// TIA Portal V16 export
// export: Created 2022-07-21T09:35:35.1718284Z, ExportSetting WithDefaults, DisplayName Totally Integrated Automation Portal, DisplayVersion V16 Update 4, DisplayName TIA Portal Version Control Interface, DisplayVersion V16 Update 2, DisplayName TIA Portal Openness, DisplayVersion V16 Update 4, DisplayName SINAMICS Startdrive Advanced, DisplayVersion V16 Update 5, DisplayName SINAMICS Startdrive G130, G150, S120, S150, SINAMICS MV, S210, DisplayVersion V16 Update 5, DisplayName SINAMICS Startdrive G110M, G120, G120C, G120D, G120P, G115D, DisplayVersion V16 Update 5, DisplayName STEP 7 Professional, DisplayVersion V16 Update 4, DisplayName STEP 7 Safety, DisplayVersion V16, DisplayName WinCC Advanced, DisplayVersion V16 Update 4
FUNCTION_BLOCK "fbKRC4ExtAut"   // FB30, LAD
TITLE = External automation handling for KUKA KRC4 / Blok obsługi trybu automatyki zewnętrznej KUKA KRC4
{ S7_Optimized_Access := 'TRUE' }
VERSION : 0.1
// stored: AutoNumber false, IsIECCheckEnabled false, IsRetainMemResEnabled false, MemoryReserve 100, SetENOAutomatically false, UDAEnableTagReadback false
   VAR_INPUT
      inRobotOutputs : "typeKRC4Outputs";   // Wejścia standardowe robota / Robot standard inputs
      inAuto : Bool;   // Zezwolenie ogólne dla robota na ruch w trybie automatycznym / Enable movement in automatic mode
      inExtReset : Bool;   // Żądanie kasowania błędów / Alarm reset requested
      inStart : Bool;   // Start programu zadanego przez PgNo / Start program selected by PgNo
      inPgNo : USInt;   // Numer programu do startu w trybie automatycznym / Program number to start in automatic mode
      inServicePos : Bool;   // Robot w poyzcji serwisowej / Robot in service position
      inClock : Bool;   // Bit zegara systemowego dla generowania zbocza sygnału / Memory clock bit for signal edge generation
   END_VAR
   VAR_OUTPUT
      ouRobotInputs : "typeKRC4Inputs";   // Wyjścia standardowe robota / Robot standard outputs
      ouStdProgSelected : Bool;   // Wybrano program standardowy / Standard program selected
      ouHomePosSelected { ExternalAccessible := 'False'; ExternalVisible := 'False'; ExternalWritable := 'False'} : Bool;   // Wybrano program "pozycja bazowa" / Home position program selected
      ouServicePosSelected { ExternalAccessible := 'False'; ExternalVisible := 'False'; ExternalWritable := 'False'} : Bool;   // Wybrano program "pozycja serwisowa" / Service position program selected
      ouBrakeTestSelected { ExternalAccessible := 'False'; ExternalVisible := 'False'; ExternalWritable := 'False'} : Bool;   // Wybrano program "test hamulców" / Brake test program selected
      ouMasterTestSelected { ExternalAccessible := 'False'; ExternalVisible := 'False'; ExternalWritable := 'False'} : Bool;   // Wybrano program "test referencji" / Reference test program selected
   END_VAR
   VAR_IN_OUT
      ioRobot : "typeRobot";
   END_VAR
   VAR
      sTONIntReset { ExternalAccessible := 'False'; ExternalVisible := 'False'; ExternalWritable := 'False'} : IEC_TIMER;   // Wewnętrzny reset (timer) / Internal reset (timer)
      sTOFHoldReset { ExternalAccessible := 'False'; ExternalVisible := 'False'; ExternalWritable := 'False'} : IEC_TIMER;   // Podtrzymanie wewnętrznego resetu (timer) / Hold internal reset (timer)
      sTONPgNoValDly { ExternalAccessible := 'False'; ExternalVisible := 'False'; ExternalWritable := 'False'} : IEC_TIMER;   // Numer programu prawidłowy (timer) / Correct program number (timer)
      sSIntPgNoPrevCycle { ExternalAccessible := 'False'; ExternalVisible := 'False'; ExternalWritable := 'False'} : USInt;   // Numer programu z poprzedniego cyklu / Previous cycle program number
      sBoPFlk { ExternalAccessible := 'False'; ExternalVisible := 'False'; ExternalWritable := 'False'} : Array[1..15] of Bool;   // Bity dla wykrywania zbocza / Edge detection bits
      sBoAutoRdy { ExternalWritable := 'False'} : Bool;   // Robot gotowy do pracy w trybie automatyki zewnętrznej / Robot ready to work in external automation mode
      sBoPgNoValid { ExternalWritable := 'False'} : Bool;   // Numer programu prawidłowy / Correct program number
      sBoExtStart { ExternalWritable := 'False'} : Bool;   // Zewnętrzny start lub kontynuacja programu / External start/continue program
      sBoMoveEnable { ExternalWritable := 'False'} : Bool;   // Ogólne zezwolenie na ruch / Movement enable
      sBoPgReset { ExternalWritable := 'False'} : Bool;   // Automatyczny reset programu / Automatic program reset
      sBoReadyForProgram { ExternalWritable := 'False'} : Bool;   // Robot gotowy do przyjęcia programu / Robot ready to receive new program
      instReset { S7_SetPoint := 'True'} : "fbReset";
   END_VAR
   VAR_TEMP
      tTrue : Bool;   // Zawsze "prawda" / Always true
      tFalse : Bool;   // Zawsze "fałsz" / Always false
      tIntResetTrigger : Bool;   // Wyzwolenie wewnętrznego resetu / Trigger internal reset
      tIntReset : Bool;   // Żądanie wewnętrznego resetu / External reset requested
      tPgNoValidDly : Bool;   // Numer programu prawidłowy (opóźniony) / Correct program number (delayed)
      tRobotInServicePosition : Bool;
   END_VAR
   VAR_TEMP   // added for the SCL form of the ladder/FBD networks
      _w1 : Bool;
      _w2 : Bool;
      _w3 : Bool;
      _w4 : Bool;
   END_VAR
BEGIN

REGION Network 1: Information / Informacja
   // EXT mode handling for KUKA KRC4 robots with brake test and reference test.
   // * Used inputs: 22
   // * Used outputs: 32
   // * Variables configuration for external automation:
   // -PGNO_TYPE = 1
   // -REFLECT_PROG_NR = 1
   // -PGNO_LENGTH = 8 (bits)
   // * Input adresses configuration in robot: as in "typeKRCInputs"
   // * Output adresses configuration in robot: as in "typeKRCOutputs"
   // 
   // !!! WARNING !!! Specify program numbers in controller constants: 
   // Robot.PgNoBrakeTest 
   // Robot.PgNoMasterTest
   // Robot.PgNoServicePos
   // Obsługa trybu EXT robotów KUKA KRC4 z obsługą testu hamulców i referencji.
   // * Liczba użwanych wejść: 22
   // * Liczba używanych wyjść: 32
   // * Konfiguracja zmiennych dla automatyki zewnętrznej:
   // - PGNO_TYPE = 1
   // - REFLECT_PROG_NR = 1
   // - PGNO_LENGTH = 8 (bitow)
   // * Konfiguracja adresów wejść w robocie: tak jak "typeKRCInputs"
   // * Konfiguracja adresów wyjść w robocie: tak jak "typeKRCOutputs"
   // 
   // !!! UWAGA !!!Należy podać numery programów w w stałych sterownika:
   // Robot.PgNoBrakeTest - test hamulców
   // Robot.PgNoMasterTest - test masteringu
   // Robot.PgNoServicePos - dojazd do pozycji serwisowej
END_REGION

REGION Network 2: Always true / Zawsze "prawda"
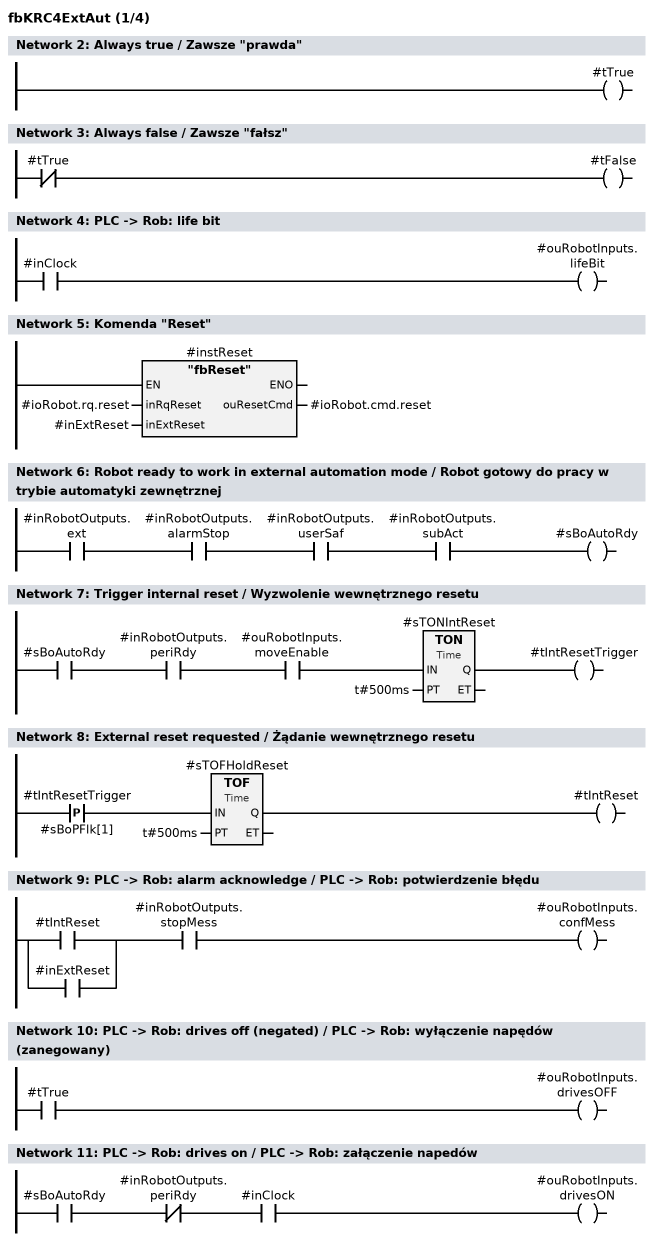
   RUNG wire#powerrail
      Coil( #tTrue )
   END_RUNG
   // the same network as SCL:
   #tTrue := TRUE;
END_REGION

REGION Network 3: Always false / Zawsze "fałsz"
   RUNG wire#powerrail
      I_Contact( #tTrue )
      Coil( #tFalse )
   END_RUNG
   // the same network as SCL:
   #tFalse := NOT #tTrue;
END_REGION

REGION Network 4: PLC -> Rob: life bit
   RUNG wire#powerrail
      Contact( #inClock )
      Coil( #ouRobotInputs.lifeBit )
   END_RUNG
   // the same network as SCL:
   #ouRobotInputs.lifeBit := #inClock;
END_REGION

REGION Network 5: Komenda "Reset"
   RUNG wire#powerrail
      #instReset(inRqReset := #ioRobot.rq.reset, inExtReset := #inExtReset, ouResetCmd => #ioRobot.cmd.reset)
   END_RUNG
   // the same network as SCL:
   #instReset(inRqReset := #ioRobot.rq.reset, inExtReset := #inExtReset, ouResetCmd => #ioRobot.cmd.reset);   // "fbReset"
END_REGION

REGION Network 6: Robot ready to work in external automation mode / Robot gotowy do pracy w trybie automatyki zewnętrznej
   RUNG wire#powerrail
      Contact( #inRobotOutputs.ext )
      Contact( #inRobotOutputs.alarmStop )
      Contact( #inRobotOutputs.userSaf )
      Contact( #inRobotOutputs.subAct )
      Coil( #sBoAutoRdy )
   END_RUNG
   // the same network as SCL:
   #sBoAutoRdy := #inRobotOutputs.ext AND #inRobotOutputs.alarmStop AND #inRobotOutputs.userSaf AND #inRobotOutputs.subAct;
END_REGION

REGION Network 7: Trigger internal reset / Wyzwolenie wewnętrznego resetu
   RUNG wire#powerrail
      Contact( #sBoAutoRdy )
      Contact( #inRobotOutputs.periRdy )
      Contact( #ouRobotInputs.moveEnable )
      { S7_Templates := "time_type := Time" } #sTONIntReset.TON(pt := t#500ms, et =>)
      Coil( #tIntResetTrigger )
   END_RUNG
   // the same network as SCL:
   #sTONIntReset.TON(IN := #sBoAutoRdy AND #inRobotOutputs.periRdy AND #ouRobotInputs.moveEnable, PT := t#500ms);
   #tIntResetTrigger := #sTONIntReset.Q;
END_REGION

REGION Network 8: External reset requested / Żądanie wewnętrznego resetu
   RUNG wire#powerrail
      P_Contact(operand := #tIntResetTrigger, bit := #sBoPFlk[1])
      { S7_Templates := "time_type := Time" } #sTOFHoldReset.TOF(pt := t#500ms, et =>)
      Coil( #tIntReset )
   END_RUNG
   // the same network as SCL:
   #_w1 := #tIntResetTrigger AND NOT #sBoPFlk[1];   // rising edge of #tIntResetTrigger
   #sBoPFlk[1] := #tIntResetTrigger;
   #sTOFHoldReset.TOF(IN := #_w1, PT := t#500ms);
   #tIntReset := #sTOFHoldReset.Q;
END_REGION

REGION Network 9: PLC -> Rob: alarm acknowledge / PLC -> Rob: potwierdzenie błędu
   RUNG wire#powerrail
      Contact( #tIntReset )
      wire#w1
      Contact( #inRobotOutputs.stopMess )
      Coil( #ouRobotInputs.confMess )
   END_RUNG
   RUNG wire#powerrail
      Contact( #inExtReset )
   END_RUNG wire#w1
   // the same network as SCL:
   #ouRobotInputs.confMess := (#tIntReset OR #inExtReset) AND #inRobotOutputs.stopMess;
END_REGION

REGION Network 10: PLC -> Rob: drives off (negated) / PLC -> Rob: wyłączenie napędów (zanegowany)
   RUNG wire#powerrail
      Contact( #tTrue )
      Coil( #ouRobotInputs.drivesOFF )
   END_RUNG
   // the same network as SCL:
   #ouRobotInputs.drivesOFF := #tTrue;
END_REGION

REGION Network 11: PLC -> Rob: drives on / PLC -> Rob: załączenie napedów
   RUNG wire#powerrail
      Contact( #sBoAutoRdy )
      I_Contact( #inRobotOutputs.periRdy )
      Contact( #inClock )
      Coil( #ouRobotInputs.drivesON )
   END_RUNG
   // the same network as SCL:
   #ouRobotInputs.drivesON := #sBoAutoRdy AND NOT #inRobotOutputs.periRdy AND #inClock;
END_REGION

REGION Network 12: PLC -> Rob: external start program / PLC -> Rob: zewnętrzny start programu
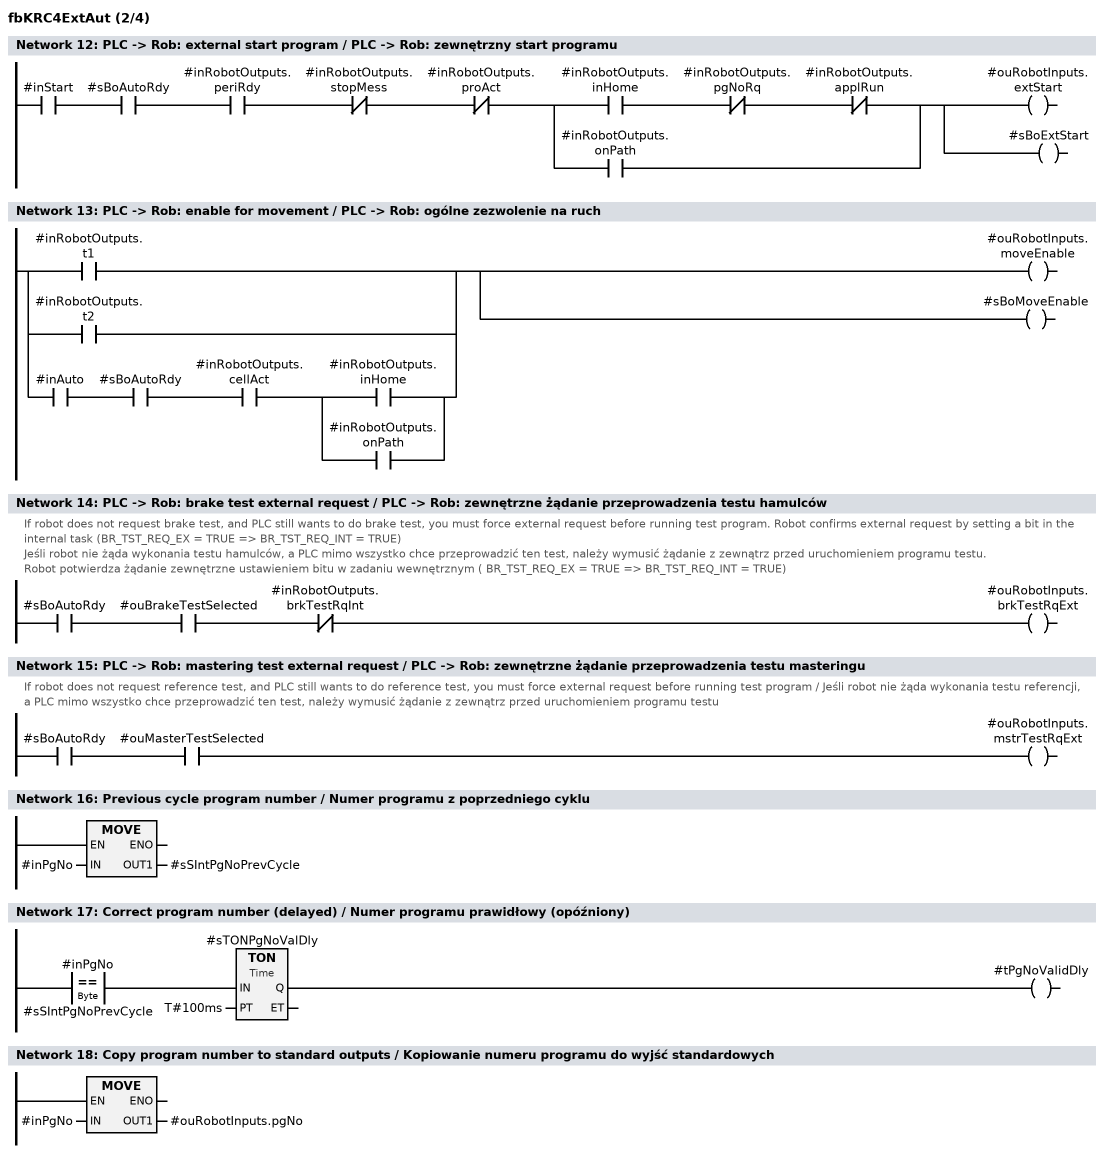
   RUNG wire#powerrail
      Contact( #inStart )
      Contact( #sBoAutoRdy )
      Contact( #inRobotOutputs.periRdy )
      I_Contact( #inRobotOutputs.stopMess )
      I_Contact( #inRobotOutputs.proAct )
      wire#w1
      Contact( #inRobotOutputs.inHome )
      I_Contact( #inRobotOutputs.pgNoRq )
      I_Contact( #inRobotOutputs.applRun )
      wire#w2
      Coil( #ouRobotInputs.extStart )
   END_RUNG
   RUNG wire#w1
      Contact( #inRobotOutputs.onPath )
   END_RUNG wire#w2
   RUNG wire#w2
      Coil( #sBoExtStart )
   END_RUNG
   // the same network as SCL:
   #ouRobotInputs.extStart := #inStart AND #sBoAutoRdy AND #inRobotOutputs.periRdy AND NOT #inRobotOutputs.stopMess AND NOT #inRobotOutputs.proAct AND ((#inRobotOutputs.inHome AND NOT #inRobotOutputs.pgNoRq AND NOT #inRobotOutputs.applRun) OR #inRobotOutputs.onPath);
   #sBoExtStart := #ouRobotInputs.extStart;
END_REGION

REGION Network 13: PLC -> Rob: enable for movement / PLC -> Rob: ogólne zezwolenie na ruch
   RUNG wire#powerrail
      Contact( #inRobotOutputs.t1 )
      wire#w1
      Coil( #ouRobotInputs.moveEnable )
   END_RUNG
   RUNG wire#powerrail
      Contact( #inRobotOutputs.t2 )
   END_RUNG wire#w1
   RUNG wire#powerrail
      Contact( #inAuto )
      Contact( #sBoAutoRdy )
      Contact( #inRobotOutputs.cellAct )
      wire#w2
      Contact( #inRobotOutputs.inHome )
   END_RUNG wire#w1
   RUNG wire#w2
      Contact( #inRobotOutputs.onPath )
   END_RUNG wire#w1
   RUNG wire#w1
      Coil( #sBoMoveEnable )
   END_RUNG
   // the same network as SCL:
   #ouRobotInputs.moveEnable := #inRobotOutputs.t1 OR #inRobotOutputs.t2 OR (#inAuto AND #sBoAutoRdy AND #inRobotOutputs.cellAct AND (#inRobotOutputs.inHome OR #inRobotOutputs.onPath));
   #sBoMoveEnable := #ouRobotInputs.moveEnable;
END_REGION

REGION Network 14: PLC -> Rob: brake test external request / PLC -> Rob: zewnętrzne żądanie przeprowadzenia testu hamulców
   // If robot does not request brake test, and PLC still wants to do brake test, you must force external request before running test program. Robot confirms external request by setting a bit in the internal task (BR_TST_REQ_EX = TRUE => BR_TST_REQ_INT = TRUE)
   // Jeśli robot nie żąda wykonania testu hamulców, a PLC mimo wszystko chce przeprowadzić ten test, należy wymusić żądanie z zewnątrz przed uruchomieniem programu testu.
   // Robot potwierdza żądanie zewnętrzne ustawieniem bitu w zadaniu wewnętrznym ( BR_TST_REQ_EX = TRUE => BR_TST_REQ_INT = TRUE)
   RUNG wire#powerrail
      Contact( #sBoAutoRdy )
      Contact( #ouBrakeTestSelected )
      I_Contact( #inRobotOutputs.brkTestRqInt )
      Coil( #ouRobotInputs.brkTestRqExt )
   END_RUNG
   // the same network as SCL:
   #ouRobotInputs.brkTestRqExt := #sBoAutoRdy AND #ouBrakeTestSelected AND NOT #inRobotOutputs.brkTestRqInt;
END_REGION

REGION Network 15: PLC -> Rob: mastering test external request / PLC -> Rob: zewnętrzne żądanie przeprowadzenia testu masteringu
   // If robot does not request reference test, and PLC still wants to do reference test, you must force external request before running test program / Jeśli robot nie żąda wykonania testu referencji, a PLC mimo wszystko chce przeprowadzić ten test, należy wymusić żądanie z zewnątrz przed uruchomieniem programu testu
   RUNG wire#powerrail
      Contact( #sBoAutoRdy )
      Contact( #ouMasterTestSelected )
      Coil( #ouRobotInputs.mstrTestRqExt )
   END_RUNG
   // the same network as SCL:
   #ouRobotInputs.mstrTestRqExt := #sBoAutoRdy AND #ouMasterTestSelected;
END_REGION

REGION Network 16: Previous cycle program number / Numer programu z poprzedniego cyklu
   RUNG wire#powerrail
      Move(in := #inPgNo, out1 => #sSIntPgNoPrevCycle)
   END_RUNG
   // the same network as SCL:
   #sSIntPgNoPrevCycle := #inPgNo;
END_REGION

REGION Network 17: Correct program number (delayed) / Numer programu prawidłowy (opóźniony)
   RUNG wire#powerrail
      { S7_Templates := "SrcType := Byte" } EQ_Contact(in1 := #inPgNo, in2 := #sSIntPgNoPrevCycle)
      { S7_Templates := "time_type := Time" } #sTONPgNoValDly.TON(pt := T#100ms, et =>)
      Coil( #tPgNoValidDly )
   END_RUNG
   // the same network as SCL:
   #sTONPgNoValDly.TON(IN := #inPgNo = #sSIntPgNoPrevCycle, PT := T#100ms);
   #tPgNoValidDly := #sTONPgNoValDly.Q;
END_REGION

REGION Network 18: Copy program number to standard outputs / Kopiowanie numeru programu do wyjść standardowych
   RUNG wire#powerrail
      Move(in := #inPgNo, out1 => #ouRobotInputs.pgNo)
   END_RUNG
   // the same network as SCL:
   #ouRobotInputs.pgNo := #inPgNo;
END_REGION

REGION Network 19: PLC -> Rob: program number - correct / PLC -> Rob: nr programu - poprawny
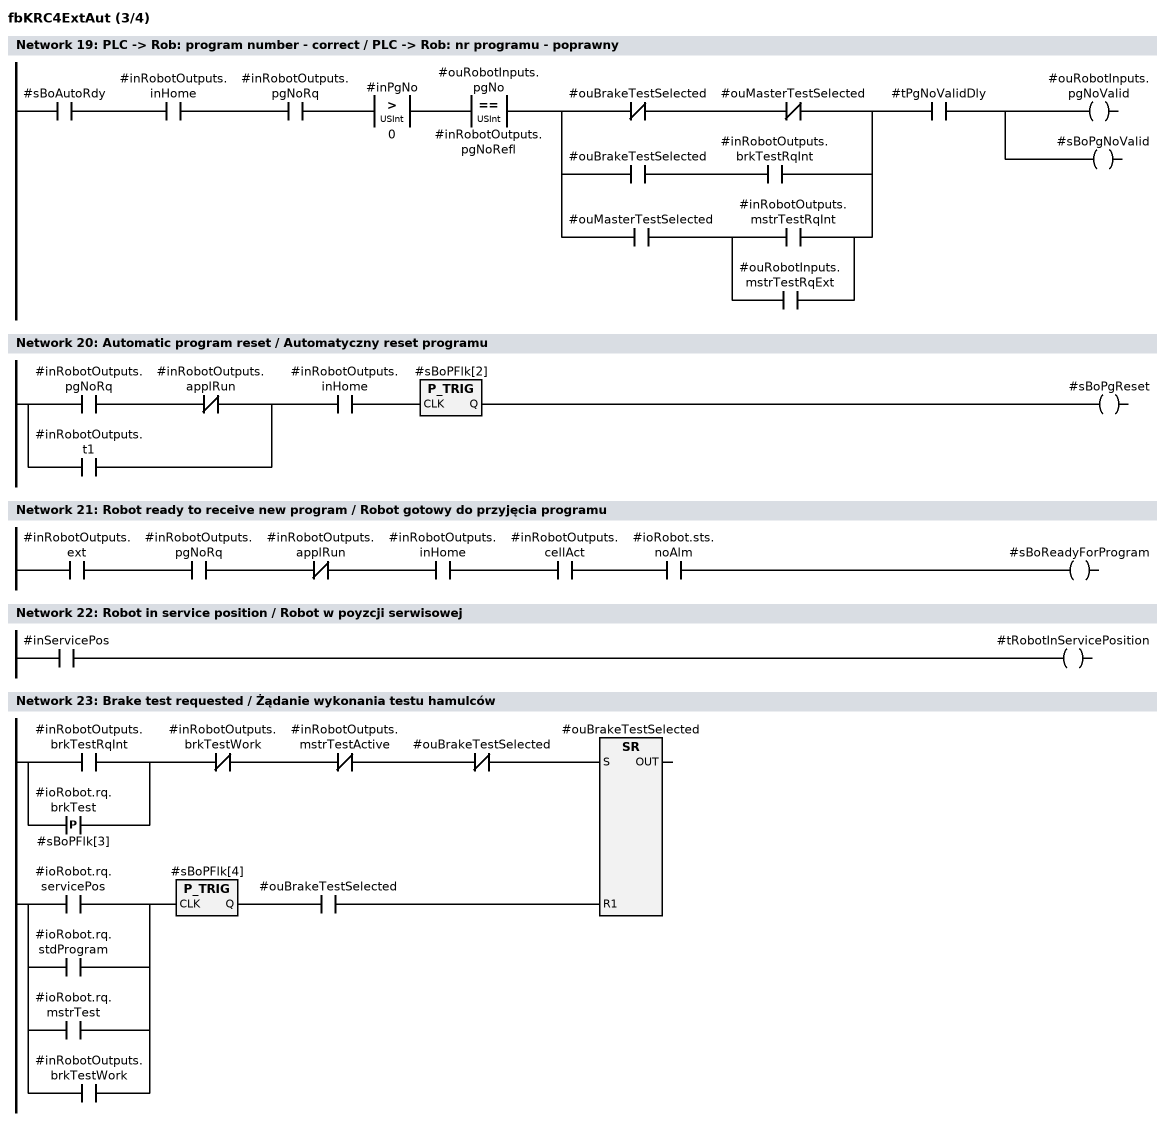
   RUNG wire#powerrail
      Contact( #sBoAutoRdy )
      Contact( #inRobotOutputs.inHome )
      Contact( #inRobotOutputs.pgNoRq )
      { S7_Templates := "SrcType := USInt" } GT_Contact(in1 := #inPgNo, in2 := 0)
      { S7_Templates := "SrcType := USInt" } EQ_Contact(in1 := #ouRobotInputs.pgNo, in2 := #inRobotOutputs.pgNoRefl)
      wire#w1
      I_Contact( #ouBrakeTestSelected )
      I_Contact( #ouMasterTestSelected )
      wire#w2
      Contact( #tPgNoValidDly )
      wire#w4
      Coil( #ouRobotInputs.pgNoValid )
   END_RUNG
   RUNG wire#w1
      Contact( #ouBrakeTestSelected )
      Contact( #inRobotOutputs.brkTestRqInt )
   END_RUNG wire#w2
   RUNG wire#w1
      Contact( #ouMasterTestSelected )
      wire#w3
      Contact( #inRobotOutputs.mstrTestRqInt )
   END_RUNG wire#w2
   RUNG wire#w3
      Contact( #ouRobotInputs.mstrTestRqExt )
   END_RUNG wire#w2
   RUNG wire#w4
      Coil( #sBoPgNoValid )
   END_RUNG
   // the same network as SCL:
   #ouRobotInputs.pgNoValid := #sBoAutoRdy AND #inRobotOutputs.inHome AND #inRobotOutputs.pgNoRq AND (#inPgNo > 0) AND (#ouRobotInputs.pgNo = #inRobotOutputs.pgNoRefl) AND ((NOT #ouBrakeTestSelected AND NOT #ouMasterTestSelected) OR (#ouBrakeTestSelected AND #inRobotOutputs.brkTestRqInt) OR (#ouMasterTestSelected AND (#inRobotOutputs.mstrTestRqInt OR #ouRobotInputs.mstrTestRqExt))) AND #tPgNoValidDly;
   #sBoPgNoValid := #ouRobotInputs.pgNoValid;
END_REGION

REGION Network 20: Automatic program reset / Automatyczny reset programu
   RUNG wire#powerrail
      Contact( #inRobotOutputs.pgNoRq )
      I_Contact( #inRobotOutputs.applRun )
      wire#w1
      Contact( #inRobotOutputs.inHome )
      P_Trig( #sBoPFlk[2] )
      Coil( #sBoPgReset )
   END_RUNG
   RUNG wire#powerrail
      Contact( #inRobotOutputs.t1 )
   END_RUNG wire#w1
   // the same network as SCL:
   #_w1 := ((#inRobotOutputs.pgNoRq AND NOT #inRobotOutputs.applRun) OR #inRobotOutputs.t1) AND #inRobotOutputs.inHome;
   #_w2 := #_w1 AND NOT #sBoPFlk[2];   // rising edge
   #sBoPFlk[2] := #_w1;
   #sBoPgReset := #_w2;
END_REGION

REGION Network 21: Robot ready to receive new program / Robot gotowy do przyjęcia programu
   RUNG wire#powerrail
      Contact( #inRobotOutputs.ext )
      Contact( #inRobotOutputs.pgNoRq )
      I_Contact( #inRobotOutputs.applRun )
      Contact( #inRobotOutputs.inHome )
      Contact( #inRobotOutputs.cellAct )
      Contact( #ioRobot.sts.noAlm )
      Coil( #sBoReadyForProgram )
   END_RUNG
   // the same network as SCL:
   #sBoReadyForProgram := #inRobotOutputs.ext AND #inRobotOutputs.pgNoRq AND NOT #inRobotOutputs.applRun AND #inRobotOutputs.inHome AND #inRobotOutputs.cellAct AND #ioRobot.sts.noAlm;
END_REGION

REGION Network 22: Robot in service position / Robot w poyzcji serwisowej
   RUNG wire#powerrail
      Contact( #inServicePos )
      Coil( #tRobotInServicePosition )
   END_RUNG
   // the same network as SCL:
   #tRobotInServicePosition := #inServicePos;
END_REGION

REGION Network 23: Brake test requested / Żądanie wykonania testu hamulców
   RUNG wire#powerrail
      Contact( #inRobotOutputs.brkTestRqInt )
      wire#w1
      I_Contact( #inRobotOutputs.brkTestWork )
      I_Contact( #inRobotOutputs.mstrTestActive )
      I_Contact( #ouBrakeTestSelected )
      S_SR(operand := #ouBrakeTestSelected, r1 := wire#w3)
   END_RUNG
   RUNG wire#powerrail
      P_Contact(operand := #ioRobot.rq.brkTest, bit := #sBoPFlk[3])
   END_RUNG wire#w1
   RUNG wire#powerrail
      Contact( #ioRobot.rq.servicePos )
      wire#w2
      P_Trig( #sBoPFlk[4] )
      Contact( #ouBrakeTestSelected )
   END_RUNG wire#w3
   RUNG wire#powerrail
      Contact( #ioRobot.rq.stdProgram )
   END_RUNG wire#w2
   RUNG wire#powerrail
      Contact( #ioRobot.rq.mstrTest )
   END_RUNG wire#w2
   RUNG wire#powerrail
      Contact( #inRobotOutputs.brkTestWork )
   END_RUNG wire#w2
   // the same network as SCL:
   #_w1 := #ioRobot.rq.brkTest AND NOT #sBoPFlk[3];   // rising edge of #ioRobot.rq.brkTest
   #sBoPFlk[3] := #ioRobot.rq.brkTest;
   #_w2 := #ioRobot.rq.servicePos OR #ioRobot.rq.stdProgram OR #ioRobot.rq.mstrTest OR #inRobotOutputs.brkTestWork;
   #_w3 := #_w2 AND NOT #sBoPFlk[4];   // rising edge
   #sBoPFlk[4] := #_w2;
   #_w4 := #_w3 AND #ouBrakeTestSelected;
   IF (#inRobotOutputs.brkTestRqInt OR #_w1) AND NOT #inRobotOutputs.brkTestWork AND NOT #inRobotOutputs.mstrTestActive AND NOT #ouBrakeTestSelected THEN
       #ouBrakeTestSelected := TRUE;   // SR flip-flop
   END_IF;
   IF #_w4 THEN #ouBrakeTestSelected := FALSE; END_IF;
END_REGION

REGION Network 24: Robot 1 request mastering test / Robot 1 żądanie wykonania testu masteringu
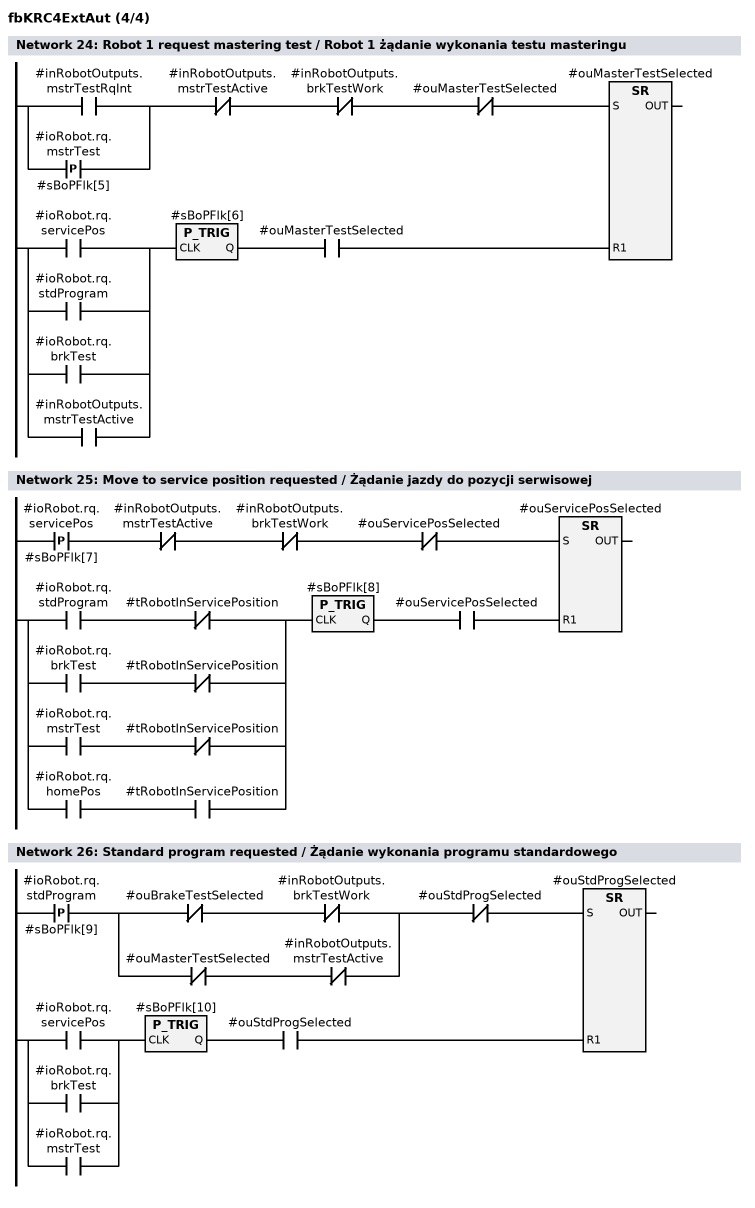
   RUNG wire#powerrail
      Contact( #inRobotOutputs.mstrTestRqInt )
      wire#w1
      I_Contact( #inRobotOutputs.mstrTestActive )
      I_Contact( #inRobotOutputs.brkTestWork )
      I_Contact( #ouMasterTestSelected )
      S_SR(operand := #ouMasterTestSelected, r1 := wire#w3)
   END_RUNG
   RUNG wire#powerrail
      P_Contact(operand := #ioRobot.rq.mstrTest, bit := #sBoPFlk[5])
   END_RUNG wire#w1
   RUNG wire#powerrail
      Contact( #ioRobot.rq.servicePos )
      wire#w2
      P_Trig( #sBoPFlk[6] )
      Contact( #ouMasterTestSelected )
   END_RUNG wire#w3
   RUNG wire#powerrail
      Contact( #ioRobot.rq.stdProgram )
   END_RUNG wire#w2
   RUNG wire#powerrail
      Contact( #ioRobot.rq.brkTest )
   END_RUNG wire#w2
   RUNG wire#powerrail
      Contact( #inRobotOutputs.mstrTestActive )
   END_RUNG wire#w2
   // the same network as SCL:
   #_w1 := #ioRobot.rq.mstrTest AND NOT #sBoPFlk[5];   // rising edge of #ioRobot.rq.mstrTest
   #sBoPFlk[5] := #ioRobot.rq.mstrTest;
   #_w2 := #ioRobot.rq.servicePos OR #ioRobot.rq.stdProgram OR #ioRobot.rq.brkTest OR #inRobotOutputs.mstrTestActive;
   #_w3 := #_w2 AND NOT #sBoPFlk[6];   // rising edge
   #sBoPFlk[6] := #_w2;
   #_w4 := #_w3 AND #ouMasterTestSelected;
   IF (#inRobotOutputs.mstrTestRqInt OR #_w1) AND NOT #inRobotOutputs.mstrTestActive AND NOT #inRobotOutputs.brkTestWork AND NOT #ouMasterTestSelected THEN
       #ouMasterTestSelected := TRUE;   // SR flip-flop
   END_IF;
   IF #_w4 THEN #ouMasterTestSelected := FALSE; END_IF;
END_REGION

REGION Network 25: Move to service position requested / Żądanie jazdy do pozycji serwisowej
   RUNG wire#powerrail
      P_Contact(operand := #ioRobot.rq.servicePos, bit := #sBoPFlk[7])
      I_Contact( #inRobotOutputs.mstrTestActive )
      I_Contact( #inRobotOutputs.brkTestWork )
      I_Contact( #ouServicePosSelected )
      S_SR(operand := #ouServicePosSelected, r1 := wire#w2)
   END_RUNG
   RUNG wire#powerrail
      Contact( #ioRobot.rq.stdProgram )
      I_Contact( #tRobotInServicePosition )
      wire#w1
      P_Trig( #sBoPFlk[8] )
      Contact( #ouServicePosSelected )
   END_RUNG wire#w2
   RUNG wire#powerrail
      Contact( #ioRobot.rq.brkTest )
      I_Contact( #tRobotInServicePosition )
   END_RUNG wire#w1
   RUNG wire#powerrail
      Contact( #ioRobot.rq.mstrTest )
      I_Contact( #tRobotInServicePosition )
   END_RUNG wire#w1
   RUNG wire#powerrail
      Contact( #ioRobot.rq.homePos )
      Contact( #tRobotInServicePosition )
   END_RUNG wire#w1
   // the same network as SCL:
   #_w1 := #ioRobot.rq.servicePos AND NOT #sBoPFlk[7];   // rising edge of #ioRobot.rq.servicePos
   #sBoPFlk[7] := #ioRobot.rq.servicePos;
   #_w2 := (#ioRobot.rq.stdProgram AND NOT #tRobotInServicePosition) OR (#ioRobot.rq.brkTest AND NOT #tRobotInServicePosition) OR (#ioRobot.rq.mstrTest AND NOT #tRobotInServicePosition) OR (#ioRobot.rq.homePos AND #tRobotInServicePosition);
   #_w3 := #_w2 AND NOT #sBoPFlk[8];   // rising edge
   #sBoPFlk[8] := #_w2;
   #_w4 := #_w3 AND #ouServicePosSelected;
   IF #_w1 AND NOT #inRobotOutputs.mstrTestActive AND NOT #inRobotOutputs.brkTestWork AND NOT #ouServicePosSelected THEN
       #ouServicePosSelected := TRUE;   // SR flip-flop
   END_IF;
   IF #_w4 THEN #ouServicePosSelected := FALSE; END_IF;
END_REGION

REGION Network 26: Standard program requested / Żądanie wykonania programu standardowego
   RUNG wire#powerrail
      P_Contact(operand := #ioRobot.rq.stdProgram, bit := #sBoPFlk[9])
      wire#w1
      I_Contact( #ouBrakeTestSelected )
      I_Contact( #inRobotOutputs.brkTestWork )
      wire#w2
      I_Contact( #ouStdProgSelected )
      S_SR(operand := #ouStdProgSelected, r1 := wire#w4)
   END_RUNG
   RUNG wire#w1
      I_Contact( #ouMasterTestSelected )
      I_Contact( #inRobotOutputs.mstrTestActive )
   END_RUNG wire#w2
   RUNG wire#powerrail
      Contact( #ioRobot.rq.servicePos )
      wire#w3
      P_Trig( #sBoPFlk[10] )
      Contact( #ouStdProgSelected )
   END_RUNG wire#w4
   RUNG wire#powerrail
      Contact( #ioRobot.rq.brkTest )
   END_RUNG wire#w3
   RUNG wire#powerrail
      Contact( #ioRobot.rq.mstrTest )
   END_RUNG wire#w3
   // the same network as SCL:
   #_w1 := #ioRobot.rq.stdProgram AND NOT #sBoPFlk[9];   // rising edge of #ioRobot.rq.stdProgram
   #sBoPFlk[9] := #ioRobot.rq.stdProgram;
   #_w2 := #ioRobot.rq.servicePos OR #ioRobot.rq.brkTest OR #ioRobot.rq.mstrTest;
   #_w3 := #_w2 AND NOT #sBoPFlk[10];   // rising edge
   #sBoPFlk[10] := #_w2;
   #_w4 := #_w3 AND #ouStdProgSelected;
   IF #_w1 AND ((NOT #ouBrakeTestSelected AND NOT #inRobotOutputs.brkTestWork) OR (NOT #ouMasterTestSelected AND NOT #inRobotOutputs.mstrTestActive)) AND NOT #ouStdProgSelected THEN
       #ouStdProgSelected := TRUE;   // SR flip-flop
   END_IF;
   IF #_w4 THEN #ouStdProgSelected := FALSE; END_IF;
END_REGION
END_FUNCTION_BLOCK
